DATA_BLOCK "ST10_Flow23_KReserveLifting_iDB"
{ S7_Optimized_Access := 'TRUE' }
VERSION : 0.1
NON_RETAIN
// ATTRIBUTES
// AUTO_NUMBER = False
// BLOCK_NUMBER = 1093
// END_ATTRIBUTES
"ST10_Flow23_KReserveLifting"

BEGIN

END_DATA_BLOCK

